Omron CX-Programmer project NewProject (CX-Programmer 9.51)

# PLC NewPLC1: CP1L L

## Global symbols (name address type ; comment)
0.00 BOOL  ; Stepper enable
0.01 BOOL  ; Start cykle
0.02 BOOL  ; Stop cykle
0.03 BOOL  ; Set F2
0.04 BOOL  ; Set F3
0.05 BOOL  ; Set F4
100.00 BOOL  ; wy1
100.01 BOOL  ; SMC81_DIR
100.02 BOOL  ; SMC81_ EN
100.03 BOOL  ; Stepper motor direction
100.04 BOOL  ; Output1
100.05 BOOL  ; Timer On
D0 CHANNEL  ; Nr Puls
T0000 BOOL  ; 2 s delay
W0 CHANNEL  ; Status
W0.01 BOOL  ; Generation
W0.03 BOOL  ; Output Coplete
W0.04 BOOL  ; Pulse Not Stop
W1.00 BOOL  ; Impuls startowy

## Program NewProgram1 (cyclic task 0)
; CX_DEMO4. Wykorzystanie funkcji SPED i PULS do sterowania silnika w trybie położenia

### Section Section1

### Section END

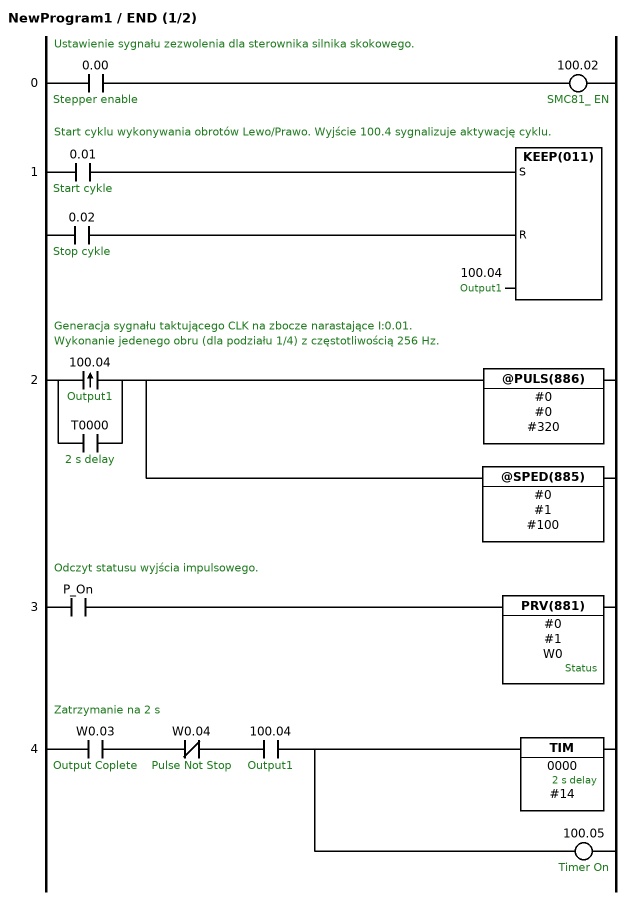
; rung 0: Ustawienie sygnału zezwolenia dla sterownika silnika skokowego.
LD 0.00  ; Stepper enable
OUT 100.02  ; SMC81_ EN
; rung 1: Start cyklu wykonywania obrotów Lewo/Prawo. Wyjście 100.4 sygnalizuje aktywację cyklu.
LD 0.01  ; Start cykle
LD 0.02  ; Stop cykle
KEEP(011) 100.04  ; Output1
; rung 2: Generacja sygnału taktującego CLK na zbocze narastające I:0.01. / Wykonanie jedenego obru (dla podziału 1/4) z częstotliwością 256 Hz.
@LD 100.04  ; Output1
OR T0000  ; 2 s delay
@PULS(886) #0 #0 #320
@SPED(885) #0 #1 #100
; rung 3: Odczyt statusu wyjścia impulsowego.
LD P_On
PRV(881) #0 #1 W0  ; Status
; rung 4: Zatrzymanie na 2 s
LD W0.03  ; Output Coplete
ANDNOT W0.04  ; Pulse Not Stop
AND 100.04  ; Output1
TIM 0000 #14  ; 2 s delay
OUT 100.05  ; Timer On

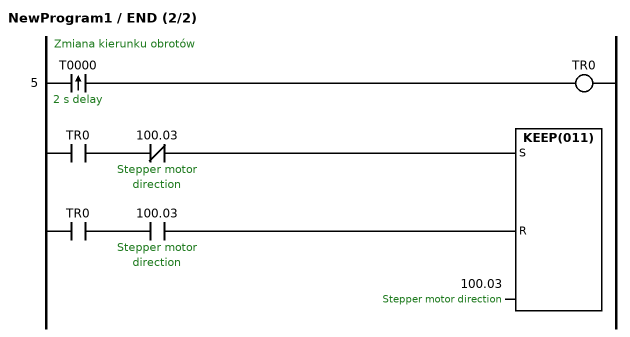
; rung 5: Zmiana kierunku obrotów
@LD T0000  ; 2 s delay
OUT TR0
ANDNOT 100.03  ; Stepper motor direction
LD TR0
AND 100.03  ; Stepper motor direction
KEEP(011) 100.03  ; Stepper motor direction
; rung 6
END(001)